PROGRAM Stn052_51_Stn126MainMergePrestop
VAR
	//correct
	{attribute 'TcLinkToOSO' := '.iPuckPresent     :=  <0,1,2>TIIB[N28S00 (AL1332)]^N28S03 (AL2341)^TxPDO^input byte 0;
								 .iBufferFull    :=  <0,1,2>TIIB[N28S00 (AL1332)]^N28S03 (AL2341)^TxPDO^input byte 2;
								 .oStopLower     :=  <0,1,1>TIIB[N28S00 (AL1332)]^N28S06 (EX260)^RxPDO^output byte 0'}	
	fbConvStop: FB_ConvStop;
END_VAR

//  This code instantiates a component that is implimented as a common function block
//    Note that I/O is linked directly to I/O variables inside the named instance

gStn052_51_Stn126MainMergePrestop.ConvRunning := gConsumed_SafetyInterfaceConv.MtrRunning.Enc054Mtr03;
 
fbConvStop(
	pStn := ADR(gStn052),
	pCmp := ADR(gStn052_51_Stn126MainMergePrestop),
	pUpstreamStop := 0,
	pStateTraceBuffer := ADR(gStn052_StateTraceBuffer),
	pStateTraceFifo := ADR(gStn052_StateTraceFifo),
	pStats := ADR(gStn052_02_Stats));

END_PROGRAM

(* stored: Version 1.1.0.1, ProductVersion 3.1.4024.6
   POU Stn052_51_Stn126MainMergePrestop: Id {e4453342-2511-4f3d-9536-daf9a75bd906}, SpecialFunc None *)
